// TIA Portal V20 export
FUNCTION "EM_Monitor" : Void   // FC32778, LAD
// stored: Namespace Unit1, SetENOAutomatically false
   VAR_INPUT
      EM_Relation : Struct
         em00 : "Unit1.type_emRelations_em0";
         em01 : "Unit1.type_emRelations_em1";
         em02 : "Unit1.type_emRelations_em2";
         em03 : "Unit1.type_emRelations_em3";
         em04 : "Unit1.type_emRelations_em4";
         em05 : "Unit1.type_emRelations_em5";
         em06 : "Unit1.type_emRelations_em6";
         em07 : "Unit1.type_emRelations_em7";
         em08 : "Unit1.type_emRelations_em8";
         em09 : "Unit1.type_emRelations_em9";
         em10 : "Unit1.type_emRelations_em10";
         em11 : "Unit1.type_emRelations_em11";
         em12 : "Unit1.type_emRelations_em12";
         em13 : "Unit1.type_emRelations_em13";
      END_STRUCT;
   END_VAR
BEGIN

REGION Network 1: **
END_REGION

REGION Network 2: EM00
END_REGION

REGION Network 3 (SCL): EM00
END_REGION

REGION Network 4: EM01
END_REGION

REGION Network 5 (SCL): EM01
END_REGION

REGION Network 6: EM02
END_REGION

REGION Network 7 (SCL): EM02
   "Unit1.EM_MotorData".DR1_JROutPP_Left_X := "Unit1.EmNodes".emRelations.em02.cmStatus.JROutPnPLeftAxisX.monitoring.actualPosition;
   "Unit1.EM_MotorData".DR2_JROutPP_Left_Z := "Unit1.EmNodes".emRelations.em02.cmStatus.JROutPnPLeftAxisZ.monitoring.actualPosition;
   "Unit1.EM_MotorData".DR3_JROutPP_Right_X := "Unit1.EmNodes".emRelations.em02.cmStatus.JROutPnPRightAxisX.monitoring.actualPosition;
   "Unit1.EM_MotorData".DR4_JROutPP_Right_Z := "Unit1.EmNodes".emRelations.em02.cmStatus.JROutPnPRightAxisZ.monitoring.actualPosition;
END_REGION

REGION Network 8: EM03
END_REGION

REGION Network 9 (SCL): EM03
   "Unit1.EM_MotorData".DR5_T_TapeAxis_X := "Unit1.EmNodes".emRelations.em03.cmStatus.TopTapeAxisX.monitoring.actualPosition;
   "Unit1.EM_MotorData".DR6_T_TapeAxis_Y := "Unit1.EmNodes".emRelations.em03.cmStatus.TopTapeAxisY.monitoring.actualPosition;
END_REGION

REGION Network 10: EM04
END_REGION

REGION Network 11 (SCL): EM04
   "Unit1.EmNodes".emRelations.em04.sequence.sideTapeLoading.jobInterface.chargeJob2.workingDone := #EM_Relation.em04.sequence.sideTapeLoading.jobInterface.chargeJob2.workingDone;
   "Unit1.EmNodes".emRelations.em04.sequence.sideTapeAttachment.jobInterface.leftTapeGetJob3.workingDone := #EM_Relation.em04.sequence.sideTapeAttachment.jobInterface.rightTapeGetJob2.workingDone;
   "Unit1.EmNodes".emRelations.em04.sequence.sideTapeAttachment.jobInterface.leftTapeGetJob3.workingDone := #EM_Relation.em04.sequence.sideTapeAttachment.jobInterface.rightTapeGetJob2.workingDone;
   "Unit1.EmNodes".emRelations.em04.sequence.sideTapeAttachment.jobInterface.tape1PutJob4.workingDone := #EM_Relation.em04.sequence.sideTapeAttachment.jobInterface.tape1PutJob4.workingDone;
   "Unit1.EmNodes".emRelations.em04.sequence.sideTapeAttachment.jobInterface.tape2PutJob5.workingDone := #EM_Relation.em04.sequence.sideTapeAttachment.jobInterface.tape2PutJob5.workingDone;

   "Unit1.EmNodes".emRelations.em04.sequence.sideTapeAttachment.jobInterface.leftTapeGetJob3.workingDone := #EM_Relation.em04.sequence.sideTapeAttachment.jobInterface.rightTapeGetJob2.workingDone;
   "Unit1.EmNodes".emRelations.em04.sequence.sideTapeAttachment.jobInterface.leftTapeGetJob3.workingDone := #EM_Relation.em04.sequence.sideTapeAttachment.jobInterface.rightTapeGetJob2.workingDone;
   "Unit1.EmNodes".emRelations.em04.sequence.sideTapeAttachment.jobInterface.leftTapeGetJob3.workingDone := #EM_Relation.em04.sequence.sideTapeAttachment.jobInterface.rightTapeGetJob2.workingDone;
   "Unit1.EmNodes".emRelations.em04.sequence.sideTapeAttachment.jobInterface.leftTapeGetJob3.workingDone := #EM_Relation.em04.sequence.sideTapeAttachment.jobInterface.rightTapeGetJob2.workingDone;

   "Unit1.EM_MotorData".DR7_S_TapeFixStage_X := "Unit1.EmNodes".emRelations.em04.cmStatus.SideTapeFixStageAxisX.monitoring.actualPosition;
   "Unit1.EM_MotorData".DR8_S_TapeFixStage_C := "Unit1.EmNodes".emRelations.em04.cmStatus.SideTapeFixStageAxisC.monitoring.actualPosition;
   "Unit1.EM_MotorData".DR9_S_Attachment_X := "Unit1.EmNodes".emRelations.em04.cmStatus.SideTapeAttachmentAxisX.monitoring.actualPosition;
   "Unit1.EM_MotorData".DR10_S_Attachment_Y := "Unit1.EmNodes".emRelations.em04.cmStatus.SideTapeAttachmentAxisY.monitoring.actualPosition;
END_REGION

REGION Network 12: EM05
END_REGION

REGION Network 13 (SCL): EM05

   "Unit1.EM_MotorData".DR12_TrPP_Left_X := "Unit1.EmNodes".emRelations.em05.cmStatus.TransferPnPLeftAxisX.monitoring.actualPosition;
   "Unit1.EM_MotorData".DR13_TrPP_Left_Y := "Unit1.EmNodes".emRelations.em05.cmStatus.TransferPnPLeftAxisY.monitoring.actualPosition;
   "Unit1.EM_MotorData".DR14_TrPP_Left_Z := "Unit1.EmNodes".emRelations.em05.cmStatus.TransferPnPLeftAxisZ.monitoring.actualPosition;
   "Unit1.EM_MotorData".DR15_TrPP_Right_X := "Unit1.EmNodes".emRelations.em05.cmStatus.TransferPnPRightAxisX.monitoring.actualPosition;
   "Unit1.EM_MotorData".DR16_TrPP_Right_Y := "Unit1.EmNodes".emRelations.em05.cmStatus.TransferPnPRightAxisY.monitoring.actualPosition;
   "Unit1.EM_MotorData".DR17_TrPP_Right_Z := "Unit1.EmNodes".emRelations.em05.cmStatus.TransferPnPRightAxisZ.monitoring.actualPosition;
END_REGION

REGION Network 14: EM06
END_REGION

REGION Network 15 (SCL): EM06
   "Unit1.EM_MonitorData".EM06.WorkDone.LoadJob2 := #EM_Relation.em06.sequence.hotPressLeft.jobInterface.loadJob2.workingDone;
   "Unit1.EM_MonitorData".EM06.WorkDone.InspectionJob3 := #EM_Relation.em06.sequence.hotPressLeft.jobInterface.inspectionJob3.workingDone;
   "Unit1.EM_MonitorData".EM06.WorkDone.UnloadJob4 := #EM_Relation.em06.sequence.hotPressLeft.jobInterface.unloadJob4.workingDone;
END_REGION

REGION Network 16: EM07
END_REGION

REGION Network 17 (SCL): EM07
   "Unit1.EM_MonitorData".EM07.WorkDone.LoadJob2 := #EM_Relation.em07.sequence.hotPressRight.jobInterface.loadJob2.workingDone;
   "Unit1.EM_MonitorData".EM07.WorkDone.InspectionJob3 := #EM_Relation.em07.sequence.hotPressRight.jobInterface.inspectionJob3.workingDone;
   "Unit1.EM_MonitorData".EM07.WorkDone.UnloadJob4 := #EM_Relation.em07.sequence.hotPressRight.jobInterface.unloadJob4.workingDone;
END_REGION

REGION Network 18: EM08
END_REGION

REGION Network 19 (SCL): EM08
   "Unit1.EM_MonitorData".EM08.WorkDone.LoadJob2 := #EM_Relation.em08.sequence.hipotThickness.jobInterface.loadJob2.workingDone;
   "Unit1.EM_MonitorData".EM08.WorkDone.InspectionJob3 := #EM_Relation.em08.sequence.hipotThickness.jobInterface.inspectionJob3.workingDone;
   "Unit1.EM_MonitorData".EM08.WorkDone.UnloadJob4 := #EM_Relation.em08.sequence.hipotThickness.jobInterface.unloadJob4.workingDone;


   "Unit1.EM_MotorData".DR11_Thickness_Z := "Unit1.EmNodes".emRelations.em08.cmStatus.ThicknessAxisZ.monitoring.actualPosition;
END_REGION

REGION Network 20: EM09
END_REGION

REGION Network 21 (SCL): EM09
   "Unit1.EM_MonitorData".EM09.WorkDone.LoadJob2 := #EM_Relation.em09.sequence.vision.jobInterface.loadJob2.workingDone;
   "Unit1.EM_MonitorData".EM09.WorkDone.InspectionJob3 := #EM_Relation.em09.sequence.vision.jobInterface.inspectionJob3.workingDone;
   "Unit1.EM_MonitorData".EM09.WorkDone.UnloadJob4 := #EM_Relation.em09.sequence.vision.jobInterface.unloadJob4.workingDone;
END_REGION

REGION Network 22: EM10
END_REGION

REGION Network 23 (SCL): EM10
   "Unit1.EM_MonitorData".EM10.WorkDone.LoadJob2 := #EM_Relation.em10.sequence.laserMark.jobInterface.loadJob2.workingDone;
   "Unit1.EM_MonitorData".EM10.WorkDone.InspectionJob3 := #EM_Relation.em10.sequence.laserMark.jobInterface.inspectionJob3.workingDone;
   "Unit1.EM_MonitorData".EM10.WorkDone.UnloadJob4 := #EM_Relation.em10.sequence.laserMark.jobInterface.unloadJob4.workingDone;
END_REGION

REGION Network 24: EM11
END_REGION

REGION Network 25 (SCL): EM11
   "Unit1.EM_MonitorData".EM11.WorkDone.LoadJob2 := #EM_Relation.em11.sequence.weightCheck.jobInterface.loadJob2.workingDone;
   "Unit1.EM_MonitorData".EM11.WorkDone.InspectionJob3 := #EM_Relation.em11.sequence.weightCheck.jobInterface.inspectionJob3.workingDone;
   "Unit1.EM_MonitorData".EM11.WorkDone.UnloadJob4 := #EM_Relation.em11.sequence.weightCheck.jobInterface.unloadJob4.workingDone;
END_REGION

REGION Network 26: EM12
END_REGION

REGION Network 27 (SCL): EM12
END_REGION

REGION Network 28: EM13
END_REGION

REGION Network 29 (SCL): EM13

   "Unit1.EM_MotorData".DR18_JRUloading_X := "Unit1.EmNodes".emRelations.em13.cmStatus.JRUnloadingPnPAxisX.monitoring.actualPosition;
   "Unit1.EM_MotorData".DR19_JRUloading_Z := "Unit1.EmNodes".emRelations.em13.cmStatus.JRUnloadingPnPAxisZ.monitoring.actualPosition;
   "Unit1.EM_MotorData".DR20_JRUloading_C := "Unit1.EmNodes".emRelations.em13.cmStatus.JRUnloadingPnPAxisC.monitoring.actualPosition;
END_REGION
END_FUNCTION
